// Block: A0302_Bordatrice_PERS

DATA_BLOCK A0302_Bordatrice_PERS
VERSION : 0.1
   NON_RETAIN
   VAR
      Par : Struct
         Ax_Man : Positioning_EPOS_Machine_Par;
         Ax_Aut : A0301_Mach_Speed_Par;
      END_STRUCT;
      Pers_Data : Struct
         EncoderAbsolute_Preset_OK : Bool;
         Persistent_ActualPosition : LReal;
      END_STRUCT;
   END_VAR

BEGIN
   // No initialization required
END_DATA_BLOCK
